(* IEC 61131-3 sources: LASAL/Class/CommandDecoder, 1 file *)

(* ---- CommandDecoder.st ---- *)
(*!
<Class
	Name               = "CommandDecoder"
	Revision           = "0.0"
	RealtimeTask       = "false"
	CyclicTask         = "false"
	BackgroundTask     = "false"
	Sigmatek           = "false"
	OSInterface        = "false"
	HighPriority       = "false"
	Automatic          = "false"
	UpdateMode         = "Prescan"
	SharedCommandTable = "true"
	Objectsize         = "(450,120)">
	<Channels>
		<Server Name="ClassSvr" Visualized="false" Initialize="false" WriteProtected="true" Retentive="false"/>
		<Server Name="PhiVal" Visualized="false" Initialize="false" WriteProtected="true" Retentive="false"/>
		<Server Name="XVal" Visualized="false" Initialize="false" WriteProtected="true" Retentive="false"/>
		<Server Name="YVal" Visualized="false" Initialize="false" WriteProtected="true" Retentive="false"/>
		<Server Name="ZVal" Visualized="false" Initialize="false" WriteProtected="true" Retentive="false"/>
		<Client Name="cLib" Required="false" Internal="false"/>
	</Channels>
</Class>
*)
CommandDecoder : CLASS
  //Servers:
	ClassSvr 	: SvrChCmd_DINT;
	XVal 	: SvrCh_DINT;
	YVal 	: SvrCh_DINT;
	ZVal 	: SvrCh_DINT;
	PhiVal 	: SvrCh_DINT;
  //Clients:
	cLib 	: CltChCmd_SigCLib;
  //Variables:
		Command : ARRAY [0..4] OF CHAR;

		X : ARRAY [0..5] OF CHAR;

		Y : ARRAY [0..5] OF CHAR;

		Z : ARRAY [0..5] OF CHAR;

		Phi : ARRAY [0..5] OF CHAR;

  //Functions:

	FUNCTION GLOBAL DecodeCommand
		VAR_INPUT
			pString 	: ^CHAR;
		END_VAR;
  //Tables:
	FUNCTION @STD
		VAR_OUTPUT
			ret_code	: CONFSTATES;
		END_VAR;
	FUNCTION GLOBAL TAB @CT_;
END_CLASS;

#pragma usingLtd SigCLib

FUNCTION GLOBAL CommandDecoder::DecodeCommand
	VAR_INPUT
		pString 	: ^CHAR;
	END_VAR
  VAR
  	counter : DINT;
    commandSize : DINT;
    parameterSize : DINT;
  END_VAR

  parameterSize := 6 + 1;

  // get first 5 values (this represents the command)
  FOR counter := 0 TO 4 BY 1 DO
    Command[counter] := (pString+counter)^;
  END_FOR;

  // get the other values depending
  // on the command (these represent the command parameters)
  if Command = "CMOVE" then
    FOR counter := 0 TO 5 BY 1 DO
      X[counter] := (pString+counter+parameterSize-1)^; //6
    END_FOR;

    FOR counter := 0 TO 5 BY 1 DO
      Y[counter] := (pString+counter+parameterSize*2-1)^; //13
    END_FOR;

    FOR counter := 0 TO 5 BY 1 DO
      Z[counter] := (pString+counter+parameterSize*3-1)^; //20
    END_FOR;

    FOR counter := 0 TO 5 BY 1 DO
      Phi[counter] := (pString+counter+parameterSize*4-1)^; //27
    END_FOR;

    XVal := cLib.AToI(ps1:=#X[0]);
    YVal := cLib.AToI(ps1:=#Y[0]);
    ZVal := cLib.AToI(ps1:=#Y[0]);
    PhiVal := cLib.AToI(ps1:=#Phi[0]);
  end_if;

END_FUNCTION
